TYPE T_FolderName : STRING[25];
END_TYPE

(* stored: Version 1.1.0.1, ProductVersion 3.1.4024.15
   DUT T_FolderName: Id {c4a41328-d043-45d5-94fa-bb780e3b190b} *)
